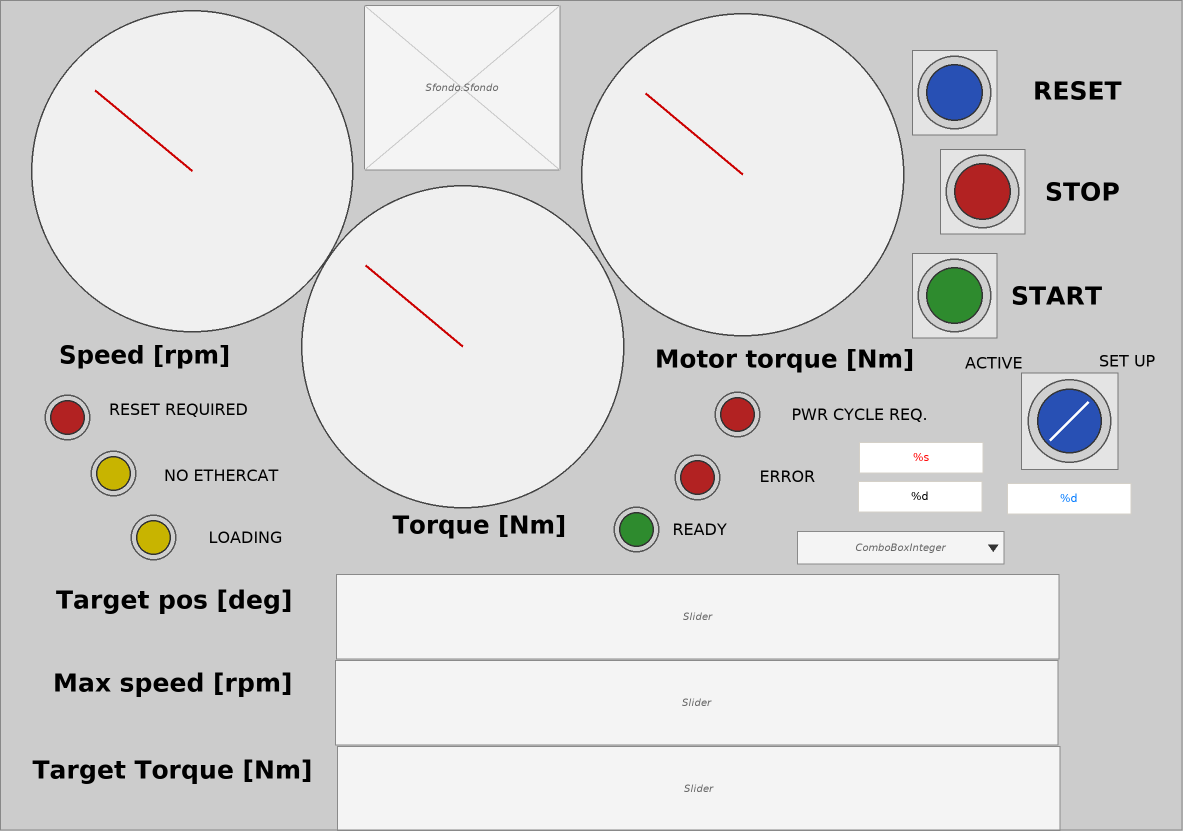
VISUALIZATION ControlPanel  // 1183x831
    Image (364,5 196x165), image: Sfondo.Sfondo
    Meter360 (300,185 325x323), value: HMI.actual_torque_nm_slow, style: Meter-Meter360-Gray, scale format: %.0f, scale -300..300
    PushSwitch (912,250 85x91), variable: CTRL.start, input disabled if: CTRL.active, behaviour: TOGGLE, style: Switch-PushSwitch-Green
    PushSwitch (937,149 91x85), variable: CTRL.stop, behaviour: TOGGLE, style: Switch-PushSwitch-Red
    Slider (335,660 723x85), variable: TRAJ.speed_selector_rpm, invisible if: CTRL.set_up, input disabled if: CTRL.set_up, scale 300..1400
    Label (31,636 284x93), "Max speed [rpm]", invisible if: CTRL.set_up
    Label (956,257 201x77), "START"
    Label (982,153 201x77), "STOP"
    Lamp1 (610,502 53x55), tooltip "WAITING", variable: CTRL.status_word.0, style: Lamp-Lamp1-Green
    Label (687,438 201x77), "ERROR"
    Label (344,502 271x46), "Torque [Nm]"
    Lamp1 (671,450 53x55), tooltip "WAITING", variable: HMI.error_light, style: Lamp-Lamp1-Red
    Label (634,491 132x77), "READY"
    Meter360 (20,10 344x322), value: HMI.actual_speed_rpm, style: Meter-Meter360-Gray, scale format: %.0f, scale -1400..1600
    Label (9,332 271x46), "Speed [rpm]"
    Meter360 (580,13 325x323), value: HMI.actual_torque_nm_fast, style: Meter-Meter360-Gray, scale format: %.1f, scale -3..3
    Label (649,336 271x46), "Motor torque [Nm]"
    PushSwitch (912,47 85x91), variable: HMI.reset_button, behaviour: TOGGLE, style: Switch-PushSwitch-Blue
    Label (977,52 201x77), "RESET"
    Lamp1 (87,446 53x55), tooltip "WAITING", variable: HMI.no_ecat_light, style: Lamp-Lamp1-Yellow
    Label (121,437 201x77), "NO ETHERCAT"
    Slider (336,574 723x85), variable: TRAJ.position_selector_deg, invisible if: CTRL.set_up, input disabled if: CTRL.set_up, scale 0..360
    Label (13,559 323x81), "Target pos [deg]", invisible if: CTRL.set_up
    ComboBoxInteger (797,531 207x33), variable: CTRL.opmode, input disabled if: CTRL.set_up, text list: 'TextList'
    Slider (337,746 723x85), variable: TRAJ.torque_selector_Nm, invisible if: CTRL.set_up, input disabled if: CTRL.set_up, scale 0..5
    Label (18,724 309x91), "Target Torque [Nm]", invisible if: CTRL.set_up
    Lamp1 (41,390 53x55), tooltip "WAITING", variable: HMI.reset_light, style: Lamp-Lamp1-Red
    Label (78,371 201x77), "RESET REQUIRED"
    Lamp1 (711,387 53x55), tooltip "WAITING", variable: HMI.out_limits_light, style: Lamp-Lamp1-Red
    Label (749,376 221x77), "PWR CYCLE REQ."
    Textfield (859,442 124x31), "%s", text variable: SDO.error_report
    RotarySwitch (1021,369 97x104), variable: CTRL.set_up, input disabled if: CTRL.wait, behaviour: TOGGLE, style: Switch-RotarySwitch-Blue
    Label (958,329 72x68), "ACTIVE"
    Label (1088,327 78x68), "SET UP"
    Lamp1 (127,510 53x55), tooltip "WAITING", variable: CTRL.wait, style: Lamp-Lamp1-Yellow
    Label (156,499 179x77), "LOADING"
    Textfield (1007,483 124x31), "%d", text variable: CTRL.status_word
    Textfield (858,481 124x31), "%d", text variable: CTRL.state_axis
END_VISUALIZATION

(* stored: Version 1.1.0.1, ProductVersion 3.1.4024.11
   Visu ControlPanel: Id {d6c62dc8-8d07-4d54-8a07-68d2dd9a1aa0} *)
